PROGRAM Bumper
VAR
	BumperStrip	AT%I*:	BOOL;
	Reset AT%I* : BOOL;
	state: Bumperstatus := Bumperstatus.init;
	Triggered AT%Q* : BOOL;
	R_Reset: R_TRIG;
	
END_VAR


CASE state OF 
	Bumperstatus.init:
		IF NOT BumperStrip AND NOT Reset THEN
			state := Bumperstatus.normal;
		END_IF	
	Bumperstatus.normal:
		IF BumperStrip THEN
			state := Bumperstatus.triggered;
			Triggered := TRUE;
		END_IF				
	Bumperstatus.triggered:
		IF NOT BumperStrip AND R_Reset.Q THEN
			state := Bumperstatus.normal;
			Triggered := FALSE;
		END_IF
END_CASE

END_PROGRAM

(* stored: Version 1.1.0.1, ProductVersion 3.1.4026.13
   POU Bumper: Id {b3b489bd-356c-424f-a2f4-3ea553d2f930}, SpecialFunc None *)
